FUNCTION_BLOCK TankCtrl_Fault EXTENDS _TankCtrl_State IMPLEMENTS I_Execute
VAR
	_exe			: Execute(THIS^);
END_VAR

METHOD Execute
VAR
	cmp		: TagCmp;
END_VAR
cmp.Set(_ctx.priv.smgr.Current);

IF NOT (_ctx.io.in.bNoWater OR _ctx.io.in.bOverload) THEN
	RETURN;
END_IF

IF cmp.Match(_ctx.state.iEStop).Match(_ctx.state.iFault).IsTrue() THEN
	RETURN;
END_IF

_ctx.priv.smgr.Request(_ctx.state.iFault);
END_METHOD

METHOD OnExecute
IF _ctx.hmi.bMultiButton THEN
	_ctx.hmi.bMultiButton := FALSE;
	
	_ctx.priv.smgr.Request(_ctx.state.iDisabled);
END_IF
END_METHOD

METHOD OnInit
_ctx.io.out.bRunPump := FALSE;

_ctx.hmi.bMultiButtonVis := TRUE;
_ctx.hmi.nMultiButtonColor := COL.Red.Raw;
_ctx.hmi.nMultiButtonText := 'Press to   Reset';

_ctx.priv.IsSystemOn.Lower();
END_METHOD

END_FUNCTION_BLOCK

(* stored: Version 1.1.0.1
   POU TankCtrl_Fault: Id {4062ce15-5d12-4b01-906c-2d981ce289b2}, SpecialFunc None
   Method Execute: Id {7f6cb2d8-4b3f-47dc-a25b-be6d1a76bbad}
   Method OnExecute: Id {f9cb5c42-c3ff-4c4f-bcc6-88a868316357}
   Method OnInit: Id {b864c809-98a7-4749-8f28-6d0bcd0c99ef} *)
